(*
	RJM Maszyny sp. z o.o.
	autor 	: Rafał Osajda
	data	: 02.02.2024
	TC		: 3.1 4024.54
	wersja	: 0.0.1.0	: pełna obsługa

	Obsługa elektrozaworu do sterowania siłownikiem pneumatycznym.sterowanie 5 na 3 2 cewki odpowietrzone
*)
FUNCTION_BLOCK FB_Electrovalve_5on3_2Coil_Vented EXTENDS FB_Electrovalve

(*
	RJM Maszyny sp. z o.o.
	autor 	: Rafał Osajda
	data	: 21.02.2024
	TC		: 3.1 4024.54
	wersja	: 0.0.1.0	: pełna obsługa

	Ustawienie odpowiednich wyjść
*)
METHOD Contol : BOOL
VAR_INPUT
	eAction									: E_ElectrovalveAction;
END_VAR
CASE eAction OF
	E_ElectrovalveAction.e_EV_Out4_Deactive	:
		bCoilA								:= FALSE;
	E_ElectrovalveAction.e_EV_OUT4_Active	:
		bCoilA								:= TRUE;
	E_ElectrovalveAction.e_EV_Out2_Deactive	:
		bCoilB								:= FALSE;
	E_ElectrovalveAction.e_EV_Out2_Active	:
		bCoilB								:= TRUE;
	E_ElectrovalveAction.e_EV_ToStart	:
		bCoilA								:= FALSE;
		bCoilB								:= TRUE;
	E_ElectrovalveAction.e_EV_ToEnd		:
		bCoilA								:= TRUE;
		bCoilB								:= FALSE;
	E_ElectrovalveAction.e_EV_Stop		:
		bCoilA								:= TRUE;
		bCoilB								:= TRUE;
	E_ElectrovalveAction.e_EV_Reset			:
		bCoilA								:= FALSE;
		bCoilB								:= FALSE;
	E_ElectrovalveAction.e_EV_Active			:
		bCoilA								:= TRUE;
		bCoilB								:= TRUE;
	E_ElectrovalveAction.e_EV_Deactive		:
		bCoilA								:= FALSE;
		bCoilB								:= FALSE;		
END_CASE
END_METHOD

METHOD FB_init : BOOL
VAR_INPUT
	bInitRetains : BOOL; // if TRUE, the retain variables are initialized (warm start / cold start)
	bInCopyCode : BOOL;  // if TRUE, the instance afterwards gets moved into the copy code (online change)
END_VAR
THIS^.eType			:= E_ElectrovalveType.C2_5na3O;
END_METHOD

END_FUNCTION_BLOCK

(* stored: Version 1.1.0.1
   POU FB_Electrovalve_5on3_2Coil_Vented: Id {794b2a56-2480-0989-026d-bc6eb7ac77ff}, SpecialFunc None
   Method Contol: Id {80410074-00ca-05c2-378d-b60c6ec1b862}
   Method FB_init: Id {babadf17-285e-4eed-8b09-470f58163602} *)
